Staubli VAL3: test.dtx

mdesc mNomSpeed
string sTest
string sTest1
